// TIA Portal project "Mypanel" (V15)
// Vorlageprojekt für das Buch mit Zielsystem S7-1200

(* hardware
DEVICE "S7-1200-Station_1"  S7-1200 Station
   slot 0: "Baugruppenträger_0"  Rack  V1.0
   slot 1: "PLC_1"  CPU 1211C DC/DC/DC  6ES7 211-1AE40-0XB0  V4.1
*)

// ===== PLC "PLC_1"  CPU 1211C DC/DC/DC =====

VAR_GLOBAL   // PLC tag table "Standard-Variablentabelle"
   "start 1" AT %E0.0 : Bool;
   "stop 1" AT %E0.1 : Bool;
   "start 2" AT %I0.2 : Bool;
   "stop 2" AT %I0.3 : Bool;
   "motor 1" AT %A0.0 : Bool;
   "motor 2" AT %Q0.1 : Bool;
   "motor 3" AT %Q0.2 : Bool;
   "motor 4" AT %Q0.3 : Bool;
   "start 3" AT %I0.4 : Bool;
   "stop 3" AT %I0.5 : Bool;
END_VAR

FUNCTION "MHJ-PLC-Lab-Function-S71200" : Void   // FC9000, SCL
{ S7_Optimized_Access := 'TRUE' }
VERSION : 0.1
   VAR_TEMP
      rdTimeReturn : Int;
      outputTime : DTL;
      SyncVal : Byte;
      forVal : Int;
      forVal_2 : Int;
      Value : Byte;
   END_VAR
   VAR CONSTANT
      CompVal : Byte := 16#34;
      Value_01 : Byte := 16#11;
      Value_01_DW : DWord := 16#A165_D992;
      Value_02_DW : DWord := 16#58BE_4401;
   END_VAR
BEGIN

   #Value:=PEEK(area := 16#82,
        dbNumber := 0,
        byteOffset := 511);
   #Value := #Value + 1;

   POKE(area := 16#82,
        dbNumber := 0,
        byteOffset := 511,
        value := #Value);

   POKE(area:=16#81,
        dbNumber:=0,
        byteOffset:=1016,
        value:=#Value_01_DW);
   POKE(area := 16#81,
        dbNumber := 0,
        byteOffset := 1020,
        value := #Value_02_DW);

   POKE(area := 16#81,
        dbNumber := 0,
        byteOffset := 511,
        value := B#16#00);

   FOR #forVal := 0 TO 120 DO
       FOR #forVal_2:=0 TO 10 DO
           #rdTimeReturn:=RD_SYS_T(#outputTime);
           #rdTimeReturn := WR_SYS_T(#outputTime);
           #rdTimeReturn := RD_SYS_T(#outputTime);
           #rdTimeReturn := WR_SYS_T(#outputTime);
       END_FOR;
       #SyncVal:= PEEK(area := 16#81,
                      dbNumber := 0,
                      byteOffset := 511);
       IF #SyncVal = #CompVal THEN
          GOTO M_1;
       END_IF;
   END_FOR;
   RETURN;

   M_1:
   POKE(area := 16#81,
        dbNumber := 0,
        byteOffset := 511,
        value := B#16#0);
END_FUNCTION

ORGANIZATION_BLOCK "Main"   // OB1, LAD, ProgramCycle
TITLE = "Main Program Sweep (Cycle)"
{ S7_Optimized_Access := 'TRUE' }
VERSION : 0.1
   VAR_INPUT
      Initial_Call : Bool;   // Initial call of this OB
      Remanence : Bool;   // =True, if remanent data are available
   END_VAR
BEGIN

REGION Network 1: Konnektierungsbaustein für PLC-Lab
   // Im Netzwerk 1 wird der Konnektierungsbaustein für PLC-Lab aufgerufen.
   // Dieser Aufruf darf nicht entfernt werden!
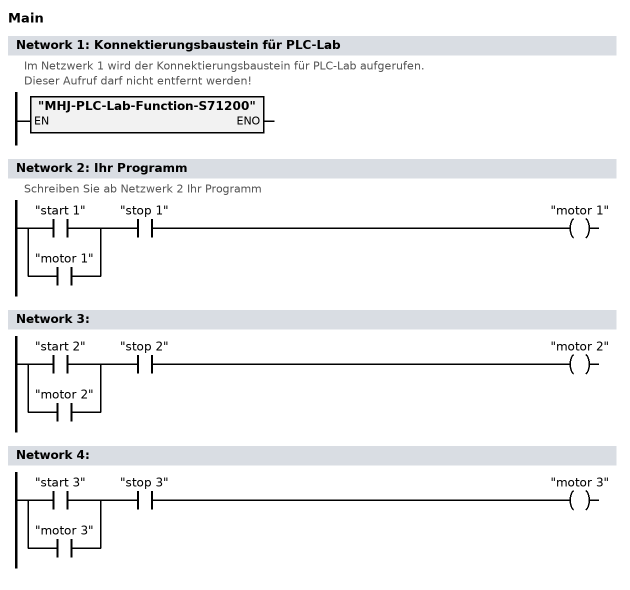
   RUNG wire#powerrail
      "MHJ-PLC-Lab-Function-S71200"()
   END_RUNG
   // the same network as SCL:
   "MHJ-PLC-Lab-Function-S71200"();
END_REGION

REGION Network 2: Ihr Programm
   // Schreiben Sie ab Netzwerk 2 Ihr Programm
   RUNG wire#powerrail
      Contact( "start 1" )
      wire#w1
      Contact( "stop 1" )
      Coil( "motor 1" )
   END_RUNG
   RUNG wire#powerrail
      Contact( "motor 1" )
   END_RUNG wire#w1
   // the same network as SCL:
   "motor 1" := ("start 1" OR "motor 1") AND "stop 1";
END_REGION

REGION Network 3
   RUNG wire#powerrail
      Contact( "start 2" )
      wire#w1
      Contact( "stop 2" )
      Coil( "motor 2" )
   END_RUNG
   RUNG wire#powerrail
      Contact( "motor 2" )
   END_RUNG wire#w1
   // the same network as SCL:
   "motor 2" := ("start 2" OR "motor 2") AND "stop 2";
END_REGION

REGION Network 4
   RUNG wire#powerrail
      Contact( "start 3" )
      wire#w1
      Contact( "stop 3" )
      Coil( "motor 3" )
   END_RUNG
   RUNG wire#powerrail
      Contact( "motor 3" )
   END_RUNG wire#w1
   // the same network as SCL:
   "motor 3" := ("start 3" OR "motor 3") AND "stop 3";
END_REGION
END_ORGANIZATION_BLOCK